Staubli VAL3: getTrackStatus.pgx

public program getTrackStatus(num& x_nTrackStatus[] (dimensions=1))
begin
  // This instruction returns the state of the last tracking move command.
  //
  // Input Param
  //  x_sConveyorList  : List of conveyors to be created
  //
  // Output param
  //  x_nTrackStatus : state of the last tracking move command
  //              0  : there is no pending tracking move command
  //              1  : a trackOn command is being executed
  //              2  : a tracking move command (linear or circular) is being executed
  //              3  : the arm is tracking a fixed point on a mobile frame
  //             -1  : the tracking is in error
  //
  //----------------------------------------------------------------
  //
  x_nTrackStatus=$trackingState()
  switch x_nTrackStatus
    case -1
      sErrorMessage=sErrMsgList[3]
    break
    case 0
      sErrorMessage=sErrMsgList[1]
    break
    case 1,2,3
      sErrorMessage=sErrMsgList[3+x_nTrackStatus]
    break
  endSwitch
end
